(* LS Electric XG5000 project: 실습1.접점 및 코일 활용하기 *)
(* PLC LSPLC *)
(* module base 0 slot 0: 입력 모듈:XGI-D21A (DC 24V 입력, 8점 (전류소스/싱크입력)) *)
(* module base 0 slot 1: 출력 모듈:XGQ-RY1A (릴레이 출력, 8점 (2A용, 단독 COM.)) *)

(* Comments on direct variables
%IX0.0.0	ON 상태일 떄 전기가 흐름
%IX0.0.1	OFF일 떄 전기가 흐름
*)

PROGRAM NewProgram (* task: 스캔 프로그램 *)
VAR
    역코일 AT %QX0.1.1 : BOOL;
    코일1 AT %QX0.1.0 : BOOL;
    코일2 AT %QX0.1.2 : BOOL;
    평상시닫힌접점 AT %IX0.0.1 : BOOL;
    평상시열린접점 AT %IX0.0.0 : BOOL;
END_VAR

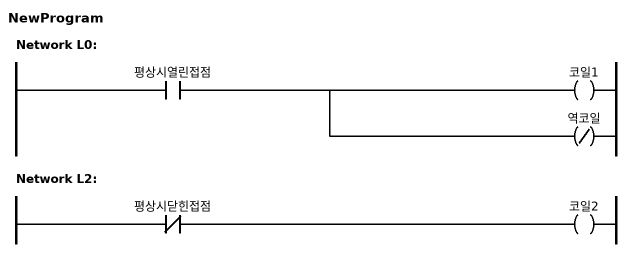
(* Rung L0 *)
코일1 := 평상시열린접점;
역코일 := NOT 평상시열린접점;
(* Rung L2 *)
코일2 := NOT 평상시닫힌접점;
END_PROGRAM